FUNCTION_BLOCK JsonDeserializer_TestSuite EXTENDS TcUnit.FB_TestSuite

TestClone();
TestReset();
TestGetArray();
TestGetKeyArray();
TestGetKeyObject();
TestGetObject();
TestTryGetBase64();
TestTryGetBoolWithFalseValue();
TestTryGetBoolWithTrueValue();
TestTryGetByte();
TestTryGetHexAsBytes();
TestTryGetDateTime();
TestTryGetDcTime();
TestTryGetDint();
TestTryGetDword();
TestTryGetFileTime();
TestTryGetInt();
TestTryGetKeyBase64();
TestTryGetKeyBoolWithFalseBoolVariable();
TestTryGetKeyBoolWithTrueBoolVariable();
TestTryGetKeyByte();
TestTryGetKeyHexAsBytes();
TestTryGetKeyDateTime();
TestTryGetKeyDcTime();
TestTryGetKeyDint();
TestTryGetKeyDword();
TestTryGetKeyFileTime();
TestTryGetKeyInt();
TestTryGetKeyLint();
TestTryGetKeyLreal();
TestTryGetKeyLtime();
TestTryGetKeyLword();
TestTryDeserializeKeyToObject();
TestTryDeserializeKeyToObjectFailsWithMissingKey();
TestTryDeserializeKeyToObjectFailsWithInvalidKey();
TestTryGetKeyReal();
TestTryGetKeySint();
TestTryGetKeyString();
TestTryGetKeyTime();
TestTryGetKeyTod();
TestTryGetKeyUdint();
TestTryGetKeyUint();
TestTryGetKeyUlint();
TestTryGetKeyUsint();
TestTryGetKeyWord();
TestTryGetLint();
TestTryGetLreal();
TestTryGetLtime();
TestTryGetLword();
TestTryDeserializeToObject();
TestTryGetReal();
TestTryGetSint();
TestTryGetString();
TestTryGetTime();
TestTryGetTod();
TestTryGetUdint();
TestTryGetUint();
TestTryGetUlint();
TestTryGetUsint();
TestTryGetWord();

METHOD PUBLIC TestClone
VAR
	jsonDeserializer : JsonDeserializer;
	clone : I_Deserializer;
    json : STRING := '{"data":100}';
    out : BYTE;
	feedback : ErrorLogger;
	hasDeserializer : BOOL;
    expected : BYTE := 100;
END_VAR
TEST('TestClone');

// add something to the original 
jsonDeserializer.TryLoad(json);

// deep clone
clone := jsonDeserializer.Clone();

// reset the original
jsonDeserializer.Reset();

// retreive the data from the clone
clone.TryGetKeyByte('data', out, feedback);

// clones are __NEW so must be disposed
clone.Dispose();

AssertEquals(
	Expected := expected,
	Actual := out,
	Message := 'Did not create a deep copy clone'
);

TEST_FINISHED();
END_METHOD

METHOD PUBLIC TestGetArray
VAR
    jsonDeserializer : JsonDeserializer;
	arrayDeserializer : I_Deserializer;
	elementDeserializer : I_Deserializer;
    json : STRING := '[100,200,300]';
    out : BYTE;
	feedback : ErrorLogger;
	hasArrayDeserializer : BOOL;
	hasElementDeserializer : BOOL;
    expected : BYTE := 100;
END_VAR
TEST('TestGetArray');

jsonDeserializer.TryLoad(json);
arrayDeserializer := jsonDeserializer.GetArray();

hasArrayDeserializer := arrayDeserializer <> 0;

IF hasArrayDeserializer THEN
	elementDeserializer := arrayDeserializer.GetElementByIndex(0);
END_IF

AssertTrue(
	Condition := hasArrayDeserializer,
	Message := 'Did not return deserializer for array'
);

hasElementDeserializer := elementDeserializer <> 0;

IF hasElementDeserializer THEN
	elementDeserializer.TryGetByte(out, feedback);
END_IF

AssertTrue(
	Condition := hasElementDeserializer,
	Message := 'Did not return deserializer for element'
);

AssertEquals(
    Expected := expected,
    Actual := out,
    Message := 'Did not produce the expected BYTE value from JSON array'
);

TEST_FINISHED();
END_METHOD

METHOD PUBLIC TestGetKeyArray
VAR
    jsonDeserializer : JsonDeserializer;
	arrayDeserializer : I_Deserializer;
	elementDeserializer : I_Deserializer;
    json : STRING := '{"myArray":[100,200,300]}';
    out : BYTE;
	feedback : ErrorLogger;
	hasArrayDeserializer : BOOL;
	hasElementDeserializer : BOOL;
    expected : BYTE := 100;
END_VAR
TEST('TestGetKeyArray');

jsonDeserializer.TryLoad(json);
arrayDeserializer := jsonDeserializer.GetKeyArray('myArray');

hasArrayDeserializer := arrayDeserializer <> 0;

IF hasArrayDeserializer THEN
	elementDeserializer := arrayDeserializer.GetElementByIndex(0);
END_IF

AssertTrue(
	Condition := hasArrayDeserializer,
	Message := 'Did not return deserializer for array'
);

hasElementDeserializer := elementDeserializer <> 0;

IF hasElementDeserializer THEN
	elementDeserializer.TryGetByte(out, feedback);
END_IF

AssertTrue(
	Condition := hasElementDeserializer,
	Message := 'Did not return deserializer for element'
);

AssertEquals(
    Expected := expected,
    Actual := out,
    Message := 'Did not produce the expected BYTE value from JSON array'
);

TEST_FINISHED();
END_METHOD

METHOD PUBLIC TestGetKeyObject
VAR
    jsonDeserializer : JsonDeserializer;
	objectDeserializer : I_Deserializer;
    json : STRING := '{"data":100}';
    out : BYTE;
	feedback : ErrorLogger;
	hasObjectDeserializer : BOOL;
    expected : BYTE := 100;
END_VAR
TEST('TestGetKeyObject');

jsonDeserializer.TryLoad(json);
objectDeserializer := jsonDeserializer.GetKeyObject('data');

hasObjectDeserializer := objectDeserializer <> 0;

IF hasObjectDeserializer THEN
	objectDeserializer.TryGetByte(out, feedback);
END_IF

AssertTrue(
	Condition := hasObjectDeserializer,
	Message := 'Did not return deserializer for object'
);

AssertEquals(
    Expected := expected,
    Actual := out,
    Message := 'Did not produce the expected BYTE value from JSON'
);

TEST_FINISHED();
END_METHOD

METHOD PUBLIC TestGetObject
VAR
    jsonDeserializer : JsonDeserializer;
	objectDeserializer : I_Deserializer;
    json : STRING := '{"data":100}';
    out : BYTE;
	feedback : ErrorLogger;
	hasObjectDeserializer : BOOL;
    expected : BYTE := 100;
END_VAR
TEST('TestGetObject');

jsonDeserializer.TryLoad(json);
objectDeserializer := jsonDeserializer.GetObject();

hasObjectDeserializer := objectDeserializer <> 0;

IF hasObjectDeserializer THEN
	objectDeserializer.TryGetKeyByte('data',out, feedback);
END_IF

AssertTrue(
	Condition := hasObjectDeserializer,
	Message := 'Did not return deserializer for object'
);

AssertEquals(
    Expected := expected,
    Actual := out,
    Message := 'Did not produce the expected BYTE value from JSON'
);

TEST_FINISHED();
END_METHOD

METHOD PUBLIC TestReset
VAR
	jsonDeserializer : JsonDeserializer;
    json : STRING := '100';
    out : BYTE;
	feedback : ErrorLogger;
    expected : BYTE := 0; 
END_VAR
TEST('TestReset');

jsonDeserializer.TryLoad(json);
jsonDeserializer.Reset();
jsonDeserializer.TryGetByte(out, feedback);

AssertEquals(
	Expected := expected,
	Actual := out,
	Message := 'Did not reset'
);

TEST_FINISHED();
END_METHOD

METHOD PUBLIC TestTryDeserializeKeyToObject
VAR
    jsonDeserializer : JsonDeserializer;
    json : STRING := '{"data":{"Name":"alice","Age":40}}';
    out : MockDeserializableUserObject;
	feedback : ErrorLogger;
    expectedName : STRING := 'alice';
	expectedAge : INT := 40;
	actualName : STRING;
	actualAge : INT;
END_VAR
TEST('TestTryDeserializeKeyToObject');
jsonDeserializer.TryLoad(json);
jsonDeserializer.TryDeserializeKeyToObject('data', out, feedback);

actualName := out.Name;
actualAge := out.Age;

AssertEquals(
    Expected := expectedName,
    Actual := actualName,
    Message := 'Did not produce the expected Object values from JSON'
);

AssertEquals(
    Expected := expectedAge,
    Actual := actualAge,
    Message := 'Did not produce the expected Object values from JSON'
);

TEST_FINISHED();
END_METHOD

METHOD PUBLIC TestTryDeserializeKeyToObjectFailsWithInvalidKey
VAR
    jsonDeserializer : JsonDeserializer;
    json : STRING := '{"data":{"Name":"alice","Age":40}}';
    out : MockDeserializableUserObject;
	feedback : ErrorLogger;
	result : BOOL;
END_VAR
TEST('TestTryDeserializeKeyToObjectFailsWithInvalidKey');
jsonDeserializer.TryLoad(json);
result := jsonDeserializer.TryDeserializeKeyToObject('', out, feedback);

AssertFalse(
	Condition := result,
	Message := 'Try returned true, even though key was invalid present');

TEST_FINISHED();
END_METHOD

METHOD PUBLIC TestTryDeserializeKeyToObjectFailsWithMissingKey
VAR
    jsonDeserializer : JsonDeserializer;
    json : STRING := '{"data":{"Name":"alice","Age":40}}';
    out : MockDeserializableUserObject;
	feedback : ErrorLogger;
	result : BOOL;
END_VAR
TEST('TestTryDeserializeKeyToObjectFailsWithMissingKey');
jsonDeserializer.TryLoad(json);
result := jsonDeserializer.TryDeserializeKeyToObject('test', out, feedback);

AssertFalse(
	Condition := result,
	Message := 'Try returned true, even though key was not present');

TEST_FINISHED();
END_METHOD

METHOD PUBLIC TestTryDeserializeToObject
VAR
    jsonDeserializer : JsonDeserializer;
    json : STRING := '{"Name":"alice","Age":40}';
    out : MockDeserializableUserObject;
	feedback : ErrorLogger;
    expectedName : STRING := 'alice';
	expectedAge : INT := 40;
	actualName : STRING;
	actualAge : INT;
END_VAR
TEST('TestTryDeserializeToObject');

jsonDeserializer.TryLoad(json);
jsonDeserializer.TryDeserializeToObject(out, feedback);

actualName := out.Name;
actualAge := out.Age;

AssertEquals(
    Expected := expectedName,
    Actual := actualName,
    Message := 'Did not produce the expected Object values from JSON'
);

AssertEquals(
    Expected := expectedAge,
    Actual := actualAge,
    Message := 'Did not produce the expected Object values from JSON'
);

TEST_FINISHED();
END_METHOD

METHOD PUBLIC TestTryGetBase64
VAR
	jsonDeserializer : JsonDeserializer;
	json : STRING := '"aGVsbG8="';
	out : ARRAY[0..4] OF BYTE;
	feedback : ErrorLogger;
	expected : ARRAY[0..4] OF BYTE := [104, 101, 108, 108, 111]; 
END_VAR
TEST('TestTryGetBase64');

jsonDeserializer.TryLoad(json);
jsonDeserializer.TryGetBase64(ADR(out), SIZEOF(out), feedback);

AssertEquals(
	Expected := expected,
	Actual := out,
	Message := 'Did not produce the expected Base64 encoded "hello" from JSON'
);

TEST_FINISHED();
END_METHOD

METHOD PUBLIC TestTryGetBoolWithFalseValue
VAR
	jsonDeserializer : JsonDeserializer;
	json : STRING := 'false';
	out : BOOL;
	feedback : ErrorLogger;
	expected : BOOL := FALSE;
END_VAR
TEST('TestTryGetBoolWithFalseValue');

jsonDeserializer.TryLoad(json);
jsonDeserializer.TryGetBool(out, feedback);

AssertEquals(
	Expected := expected,
	Actual := out,
	Message := 'Did not produce the expected JSON string for a false value'
);

TEST_FINISHED();
END_METHOD

METHOD PUBLIC TestTryGetBoolWithTrueValue
VAR
    jsonDeserializer : JsonDeserializer;
    json : STRING := 'true';
    out : BOOL;
	feedback : ErrorLogger;
    expected : BOOL := TRUE; 
END_VAR
TEST('TestTryGetBoolWithTrueValue');

jsonDeserializer.TryLoad(json);
jsonDeserializer.TryGetBool(out, feedback);

AssertEquals(
    Expected := expected,
    Actual := out,
    Message := 'Did not produce the expected true value from JSON'
);

TEST_FINISHED();
END_METHOD

METHOD PUBLIC TestTryGetByte
VAR
    jsonDeserializer : JsonDeserializer;
    json : STRING := '100';
    out : BYTE;
	feedback : ErrorLogger;
    expected : BYTE := 100; 
END_VAR
TEST('TestTryGetByte');

jsonDeserializer.TryLoad(json);
jsonDeserializer.TryGetByte(out, feedback);

AssertEquals(
    Expected := expected,
    Actual := out,
    Message := 'Did not produce the expected BYTE value from JSON'
);

TEST_FINISHED();
END_METHOD

METHOD PUBLIC TestTryGetDateTime
VAR
    jsonDeserializer : JsonDeserializer;
    json : STRING := '"2023-12-30T15:20:00"';
    out : DATE_AND_TIME;
	feedback : ErrorLogger;
    expected : DATE_AND_TIME := DT#2023-12-30-15:20:00; 
END_VAR
TEST('TestTryGetDateTime');

jsonDeserializer.TryLoad(json);
jsonDeserializer.TryGetDateTime(out, feedback);

AssertEquals(
    Expected := expected,
    Actual := out,
    Message := 'Did not produce the expected DATE_AND_TIME value from JSON'
);

TEST_FINISHED();
END_METHOD

METHOD PUBLIC TestTryGetDcTime
VAR
    jsonDeserializer : JsonDeserializer;
    json : STRING := '"2000-01-01T00:00:00.012345678"';
    out : DCTIME;
	feedback : ErrorLogger;
    expected : DCTIME := 12345678;
END_VAR
TEST('TestTryGetDcTime');

jsonDeserializer.TryLoad(json);
jsonDeserializer.TryGetDcTime(out, feedback);

AssertEquals(
    Expected := expected,
    Actual := out,
    Message := 'Did not produce the expected DCTIME value from JSON string'
);

TEST_FINISHED();
END_METHOD

METHOD PUBLIC TestTryGetDint
VAR
    jsonDeserializer : JsonDeserializer;
    json : STRING := '12345';
    out : DINT;
	feedback : ErrorLogger;
    expected : DINT := 12345;
END_VAR
TEST('TestTryGetDint');

jsonDeserializer.TryLoad(json);
jsonDeserializer.TryGetDint(out, feedback);

AssertEquals(
    Expected := expected,
    Actual := out,
    Message := 'Did not produce the expected DINT value from JSON'
);

TEST_FINISHED();
END_METHOD

METHOD PUBLIC TestTryGetDword
VAR
    jsonDeserializer : JsonDeserializer;
    json : STRING := '12345';
    out : DWORD;
	feedback : ErrorLogger;
    expected : DWORD := 12345;
END_VAR
TEST('TestTryGetDword');

jsonDeserializer.TryLoad(json);
jsonDeserializer.TryGetDword(out, feedback);

AssertEquals(
    Expected := expected,
    Actual := out,
    Message := 'Did not produce the expected DWORD value from JSON'
);

TEST_FINISHED();
END_METHOD

METHOD PUBLIC TestTryGetFileTime
VAR
    jsonDeserializer : JsonDeserializer;
    json : STRING := '"1601-01-01T00:00:01.2345678"';
    out : FILETIME;
	feedback : ErrorLogger;
    expected : FILETIME := 12345678; 
END_VAR
TEST('TestTryGetFileTime');

jsonDeserializer.TryLoad(json);
jsonDeserializer.TryGetFileTime(out, feedback);

AssertEquals(
    Expected := expected,
    Actual := out,
    Message := 'Did not produce the expected FILETIME value from JSON'
);

TEST_FINISHED();
END_METHOD

METHOD PUBLIC TestTryGetHexAsBytes
VAR
    jsonDeserializer : JsonDeserializer;
    json : STRING := '"baadf00d"';
    out : ARRAY[0..3] OF BYTE;
	feedback : ErrorLogger;
    expected : ARRAY[0..3] OF BYTE := [16#BA, 16#AD, 16#F0, 16#0D];
END_VAR
TEST('TestTryGetHexAsBytes');

jsonDeserializer.TryLoad(json);
jsonDeserializer.TryGetHexAsBytes(ADR(out), SIZEOF(out), feedback);

AssertEquals(
    Expected := expected,
    Actual := out,
    Message := 'Did not produce the expected binary data from JSON hexadecimal string'
);

TEST_FINISHED();
END_METHOD

METHOD PUBLIC TestTryGetInt
VAR
    jsonDeserializer : JsonDeserializer;
    json : STRING := '12345';
    out : INT;
	feedback : ErrorLogger;
    expected : INT := 12345;
END_VAR
TEST('TestTryGetInt');

jsonDeserializer.TryLoad(json);
jsonDeserializer.TryGetInt(out, feedback);

AssertEquals(
    Expected := expected,
    Actual := out,
    Message := 'Did not produce the expected INT value from JSON'
);

TEST_FINISHED();
END_METHOD

METHOD PUBLIC TestTryGetKeyBase64
VAR
    jsonDeserializer : JsonDeserializer;
    json : STRING := '{"data":"aGVsbG8="}';
    out : ARRAY[0..4] OF BYTE;
	feedback : ErrorLogger;
    expected : ARRAY[0..4] OF BYTE := [104, 101, 108, 108, 111];
END_VAR
TEST('TestTryGetKeyBase64');

jsonDeserializer.TryLoad(json);
jsonDeserializer.TryGetKeyBase64('data', ADR(out), SIZEOF(out), feedback);

AssertEquals(
    Expected := expected,
    Actual := out,
    Message := 'Did not produce the expected binary data from JSON Base64 encoded "hello"'
);

TEST_FINISHED();
END_METHOD

METHOD PUBLIC TestTryGetKeyBoolWithFalseBoolVariable
VAR
    jsonDeserializer : JsonDeserializer;
    json : STRING := '{"data":false}';
    out : BOOL;
	feedback : ErrorLogger;
    expected : BOOL := FALSE;
END_VAR
TEST('TestTryGetKeyBoolWithFalseBoolVariable');

jsonDeserializer.TryLoad(json);
jsonDeserializer.TryGetKeyBool('data', out, feedback);

AssertEquals(
    Expected := expected,
    Actual := out,
    Message := 'Did not produce the expected boolean value from JSON for a false value'
);

TEST_FINISHED();
END_METHOD

METHOD PUBLIC TestTryGetKeyBoolWithTrueBoolVariable
VAR
    jsonDeserializer : JsonDeserializer;
    json : STRING := '{"data":true}';
    out : BOOL;
	feedback : ErrorLogger;
    expected : BOOL := TRUE;
END_VAR
TEST('TestTryGetKeyBoolWithTrueBoolVariable');

jsonDeserializer.TryLoad(json);
jsonDeserializer.TryGetKeyBool('data', out, feedback);

AssertEquals(
    Expected := expected,
    Actual := out,
    Message := 'Did not produce the expected boolean value from JSON for a true value'
);

TEST_FINISHED();
END_METHOD

METHOD PUBLIC TestTryGetKeyByte
VAR
    jsonDeserializer : JsonDeserializer;
    json : STRING := '{"data":100}';
    out : BYTE;
	feedback : ErrorLogger;
    expected : BYTE := 100;
END_VAR
TEST('TestTryGetKeyByte');

jsonDeserializer.TryLoad(json);
jsonDeserializer.TryGetKeyByte('data', out, feedback);

AssertEquals(
    Expected := expected,
    Actual := out,
    Message := 'Did not produce the expected BYTE value from JSON'
);

TEST_FINISHED();
END_METHOD

METHOD PUBLIC TestTryGetKeyDateTime
VAR
    jsonDeserializer : JsonDeserializer;
    json : STRING := '{"data":"2023-12-30T15:20:00"}';
    out : DATE_AND_TIME;
	feedback : ErrorLogger;
    expected : DATE_AND_TIME := DT#2023-12-30-15:20:00;
END_VAR
TEST('TestTryGetKeyDateTime');

jsonDeserializer.TryLoad(json);
jsonDeserializer.TryGetKeyDateTime('data', out, feedback);

AssertEquals(
    Expected := expected,
    Actual := out,
    Message := 'Did not produce the expected DATE_AND_TIME value from JSON'
);

TEST_FINISHED();
END_METHOD

METHOD PUBLIC TestTryGetKeyDcTime
VAR
    jsonDeserializer : JsonDeserializer;
    json : STRING := '{"data":"2000-01-01T00:00:00.012345678"}';
    out : DCTIME;
	feedback : ErrorLogger;
    expected : DCTIME := 12345678;
END_VAR
TEST('TestTryGetKeyDcTime');

jsonDeserializer.TryLoad(json);
jsonDeserializer.TryGetKeyDcTime('data', out, feedback);

AssertEquals(
    Expected := expected,
    Actual := out,
    Message := 'Did not produce the expected DCTIME value from JSON string'
);

TEST_FINISHED();
END_METHOD

METHOD PUBLIC TestTryGetKeyDint
VAR
    jsonDeserializer : JsonDeserializer;
    json : STRING := '{"data":12345}';
    out : DINT;
	feedback : ErrorLogger;
    expected : DINT := 12345;
END_VAR
TEST('TestTryGetKeyDint');

jsonDeserializer.TryLoad(json);
jsonDeserializer.TryGetKeyDint('data', out, feedback);

AssertEquals(
    Expected := expected,
    Actual := out,
    Message := 'Did not produce the expected DINT value from JSON'
);

TEST_FINISHED();
END_METHOD

METHOD PUBLIC TestTryGetKeyDword
VAR
    jsonDeserializer : JsonDeserializer;
    json : STRING := '{"data":12345}';
    out : DWORD;
	feedback : ErrorLogger;
    expected : DWORD := 12345;
END_VAR
TEST('TestTryGetKeyDword');

jsonDeserializer.TryLoad(json);
jsonDeserializer.TryGetKeyDword('data', out, feedback);

AssertEquals(
    Expected := expected,
    Actual := out,
    Message := 'Did not produce the expected DWORD value from JSON'
);

TEST_FINISHED();
END_METHOD

METHOD PUBLIC TestTryGetKeyFileTime
VAR
    jsonDeserializer : JsonDeserializer;
    json : STRING := '{"data":"1601-01-01T00:00:01.2345678"}';
    out : FILETIME;
	feedback : ErrorLogger;
    expected : FILETIME := 12345678;
END_VAR
TEST('TestTryGetKeyFileTime');

jsonDeserializer.TryLoad(json);
jsonDeserializer.TryGetKeyFileTime('data', out, feedback);

AssertEquals(
    Expected := expected,
    Actual := out,
    Message := 'Did not produce the expected FILETIME value from JSON string'
);

TEST_FINISHED();
END_METHOD

METHOD PUBLIC TestTryGetKeyHexAsBytes
VAR
    jsonDeserializer : JsonDeserializer;
    json : STRING := '{"data":"baadf00d"}';
    out : ARRAY[0..3] OF BYTE;
	feedback : ErrorLogger;
    expected : ARRAY[0..3] OF BYTE := [16#BA, 16#AD, 16#F0, 16#0D];
END_VAR
TEST('TestTryGetKeyHexAsBytes');

jsonDeserializer.TryLoad(json);
jsonDeserializer.TryGetKeyHexAsBytes('data', ADR(out), SIZEOF(out), feedback);

AssertEquals(
    Expected := expected,
    Actual := out,
    Message := 'Did not produce the expected binary data from JSON hexadecimal string'
);

TEST_FINISHED();
END_METHOD

METHOD PUBLIC TestTryGetKeyInt
VAR
    jsonDeserializer : JsonDeserializer;
    json : STRING := '{"data":12345}';
    out : INT;
	feedback : ErrorLogger;
    expected : INT := 12345;
END_VAR
TEST('TestTryGetKeyInt');

jsonDeserializer.TryLoad(json);
jsonDeserializer.TryGetKeyInt('data', out, feedback);

AssertEquals(
    Expected := expected,
    Actual := out,
    Message := 'Did not produce the expected INT value from JSON'
);

TEST_FINISHED();
END_METHOD

METHOD PUBLIC TestTryGetKeyLint
VAR
    jsonDeserializer : JsonDeserializer;
    json : STRING := '{"data":9223372036854775807}';
    out : LINT;
	feedback : ErrorLogger;
    expected : LINT := 9223372036854775807;
END_VAR
TEST('TestTryGetKeyLint');

jsonDeserializer.TryLoad(json);
jsonDeserializer.TryGetKeyLint('data', out, feedback);

AssertEquals(
    Expected := expected,
    Actual := out,
    Message := 'Did not produce the expected LINT value from JSON'
);

TEST_FINISHED();
END_METHOD

METHOD PUBLIC TestTryGetKeyLreal
VAR
    jsonDeserializer : JsonDeserializer;
    json : STRING := '{"data":123456.789}';
    out : LREAL;
	feedback : ErrorLogger;
    expected : LREAL := 123456.789;
END_VAR
TEST('TestTryGetKeyLreal');

jsonDeserializer.TryLoad(json);
jsonDeserializer.TryGetKeyLreal('data', out, feedback);

AssertEquals(
    Expected := expected,
    Actual := out,
    Message := 'Did not produce the expected LREAL value from JSON'
);

TEST_FINISHED();
END_METHOD

METHOD PUBLIC TestTryGetKeyLtime
VAR
    jsonDeserializer : JsonDeserializer;
    json : STRING := '{"data":"LTIME#100d2h30m40s500ms600us700ns"}';
    out : LTIME;
	feedback : ErrorLogger;
    expected : LTIME := LTIME#100D2H30M40S500MS600US700NS;
END_VAR
TEST('TestTryGetKeyLtime');

jsonDeserializer.TryLoad(json);
jsonDeserializer.TryGetKeyLtime('data', out, feedback);

AssertEquals(
    Expected := expected,
    Actual := out,
    Message := 'Did not produce the expected LTIME value from JSON string'
);

TEST_FINISHED();
END_METHOD

METHOD PUBLIC TestTryGetKeyLword
VAR
    jsonDeserializer : JsonDeserializer;
    json : STRING := '{"data":9223372036854775807}';
    out : LWORD;
	feedback : ErrorLogger;
    expected : LWORD := 9223372036854775807;
END_VAR
TEST('TestTryGetKeyLword');

jsonDeserializer.TryLoad(json);
jsonDeserializer.TryGetKeyLword('data', out, feedback);

AssertEquals(
    Expected := expected,
    Actual := out,
    Message := 'Did not produce the expected LWORD value from JSON'
);

TEST_FINISHED();
END_METHOD

METHOD PUBLIC TestTryGetKeyReal
VAR
    jsonDeserializer : JsonDeserializer;
    json : STRING := '{"data":123.4}';
    out : REAL;
	feedback : ErrorLogger;
    expected : REAL := 123.4;
END_VAR
TEST('TestTryGetKeyReal');

jsonDeserializer.TryLoad(json);
jsonDeserializer.TryGetKeyReal('data', out, feedback);

AssertEquals(
    Expected := expected,
    Actual := out,
    Message := 'Did not produce the expected REAL value from JSON'
);

TEST_FINISHED();
END_METHOD

METHOD PUBLIC TestTryGetKeySint
VAR
    jsonDeserializer : JsonDeserializer;
    json : STRING := '{"data":123}';
    out : SINT;
	feedback : ErrorLogger;
    expected : SINT := 123;
END_VAR
TEST('TestTryGetKeySint');

jsonDeserializer.TryLoad(json);
jsonDeserializer.TryGetKeySint('data', out, feedback);

AssertEquals(
    Expected := expected,
    Actual := out,
    Message := 'Did not produce the expected SINT value from JSON'
);

TEST_FINISHED();
END_METHOD

METHOD PUBLIC TestTryGetKeyString
VAR
    jsonDeserializer : JsonDeserializer;
    json : STRING := '{"data":"foobar"}';
    out : STRING;
	feedback : ErrorLogger;
    expected : STRING := 'foobar';
END_VAR
TEST('TestTryGetKeyString');

jsonDeserializer.TryLoad(json);
jsonDeserializer.TryGetKeyString('data', out, feedback);

AssertEquals(
    Expected := expected,
    Actual := out,
    Message := 'Did not produce the expected STRING value from JSON'
);

TEST_FINISHED();
END_METHOD

METHOD PUBLIC TestTryGetKeyTime
VAR
    jsonDeserializer : JsonDeserializer;
    json : STRING := '{"data":"T#49d17h2m47s295ms"}';
    out : TIME;
	feedback : ErrorLogger;
    expected : TIME := T#49D17H2M47S295MS;
END_VAR
TEST('TestTryGetKeyTime');

jsonDeserializer.TryLoad(json);
jsonDeserializer.TryGetKeyTime('data', out, feedback);

AssertEquals(
    Expected := expected,
    Actual := out,
    Message := 'Did not produce the expected TIME value from JSON'
);

TEST_FINISHED();
END_METHOD

METHOD PUBLIC TestTryGetKeyTod
VAR
    jsonDeserializer : JsonDeserializer;
    json : STRING := '{"data":"TOD#23:01:23.456"}';
    out : TOD;
	feedback : ErrorLogger;
    expected : TOD := TOD#23:01:23.456;
END_VAR
TEST('TestTryGetKeyTod');

jsonDeserializer.TryLoad(json);
jsonDeserializer.TryGetKeyTod('data', out, feedback);

AssertEquals(
    Expected := expected,
    Actual := out,
    Message := 'Did not produce the expected TOD value from JSON'
);

TEST_FINISHED();
END_METHOD

METHOD PUBLIC TestTryGetKeyUdint
VAR
    jsonDeserializer : JsonDeserializer;
    json : STRING := '{"data":123456}';
    out : UDINT;
	feedback : ErrorLogger;
    expected : UDINT := 123456;
END_VAR
TEST('TestTryGetKeyUdint');

jsonDeserializer.TryLoad(json);
jsonDeserializer.TryGetKeyUdint('data', out, feedback);

AssertEquals(
    Expected := expected,
    Actual := out,
    Message := 'Did not produce the expected UDINT value from JSON'
);

TEST_FINISHED();
END_METHOD

METHOD PUBLIC TestTryGetKeyUint
VAR
    jsonDeserializer : JsonDeserializer;
    json : STRING := '{"data":12345}';
    out : UINT;
	feedback : ErrorLogger;
    expected : UINT := 12345;
END_VAR
TEST('TestTryGetKeyUint');

jsonDeserializer.TryLoad(json);
jsonDeserializer.TryGetKeyUint('data', out, feedback);

AssertEquals(
    Expected := expected,
    Actual := out,
    Message := 'Did not produce the expected UINT value from JSON'
);

TEST_FINISHED();
END_METHOD

METHOD PUBLIC TestTryGetKeyUlint
VAR
    jsonDeserializer : JsonDeserializer;
    json : STRING := '{"data":9223372036854775807}';
    out : ULINT;
	feedback : ErrorLogger;
    expected : ULINT := 9223372036854775807;
END_VAR
TEST('TestTryGetKeyUlint');

jsonDeserializer.TryLoad(json);
jsonDeserializer.TryGetKeyUlint('data', out, feedback);

AssertEquals(
    Expected := expected,
    Actual := out,
    Message := 'Did not produce the expected ULINT value from JSON'
);

TEST_FINISHED();
END_METHOD

METHOD PUBLIC TestTryGetKeyUsint
VAR
    jsonDeserializer : JsonDeserializer;
    json : STRING := '{"data":123}';
    out : USINT;
	feedback : ErrorLogger;
    expected : USINT := 123;
END_VAR
TEST('TestTryGetKeyUsint');

jsonDeserializer.TryLoad(json);
jsonDeserializer.TryGetKeyUsint('data', out, feedback);

AssertEquals(
    Expected := expected,
    Actual := out,
    Message := 'Did not produce the expected USINT value from JSON'
);

TEST_FINISHED();
END_METHOD

METHOD PUBLIC TestTryGetKeyWord
VAR
    jsonDeserializer : JsonDeserializer;
    json : STRING := '{"data":12345}';
    out : WORD;
	feedback : ErrorLogger;
    expected : WORD := 12345;
END_VAR
TEST('TestTryGetKeyWord');

jsonDeserializer.TryLoad(json);
jsonDeserializer.TryGetKeyWord('data', out, feedback);

AssertEquals(
    Expected := expected,
    Actual := out,
    Message := 'Did not produce the expected WORD value from JSON'
);

TEST_FINISHED();
END_METHOD

METHOD PUBLIC TestTryGetLint
VAR
    jsonDeserializer : JsonDeserializer;
    json : STRING := '9223372036854775807';
    out : LINT;
	feedback : ErrorLogger;
    expected : LINT := 9223372036854775807;
END_VAR
TEST('TestTryGetLint');

jsonDeserializer.TryLoad(json);
jsonDeserializer.TryGetLint(out, feedback);

AssertEquals(
    Expected := expected,
    Actual := out,
    Message := 'Did not produce the expected LINT value from JSON'
);

TEST_FINISHED();
END_METHOD

METHOD PUBLIC TestTryGetLreal
VAR
    jsonDeserializer : JsonDeserializer;
    json : STRING := '123456.789';
    out : LREAL;
	feedback : ErrorLogger;
    expected : LREAL := 123456.789;
END_VAR
TEST('TestTryGetLreal');

jsonDeserializer.TryLoad(json);
jsonDeserializer.TryGetLreal(out, feedback);

AssertEquals(
    Expected := expected,
    Actual := out,
    Message := 'Did not produce the expected LREAL value from JSON'
);

TEST_FINISHED();
END_METHOD

METHOD PUBLIC TestTryGetLtime
VAR
    jsonDeserializer : JsonDeserializer;
    json : STRING := '"LTIME#100d2h30m40s500ms600us700ns"';
    out : LTIME;
	feedback : ErrorLogger;
    expected : LTIME := LTIME#100D2H30M40S500MS600US700NS;
END_VAR
TEST('TestTryGetLtime');

jsonDeserializer.TryLoad(json);
jsonDeserializer.TryGetLtime(out, feedback);

AssertEquals(
    Expected := expected,
    Actual := out,
    Message := 'Did not produce the expected LTIME value from JSON string'
);

TEST_FINISHED();
END_METHOD

METHOD PUBLIC TestTryGetLword
VAR
    jsonDeserializer : JsonDeserializer;
    json : STRING := '9223372036854775807';
    out : LWORD;
	feedback : ErrorLogger;
    expected : LWORD := 9223372036854775807;
END_VAR
TEST('TestTryGetLword');

jsonDeserializer.TryLoad(json);
jsonDeserializer.TryGetLword(out, feedback);

AssertEquals(
    Expected := expected,
    Actual := out,
    Message := 'Did not produce the expected LWORD value from JSON'
);

TEST_FINISHED();
END_METHOD

METHOD PUBLIC TestTryGetReal
VAR
    jsonDeserializer : JsonDeserializer;
    json : STRING := '123.4';
    out : REAL;
	feedback : ErrorLogger;
    expected : REAL := 123.4;
END_VAR
TEST('TestTryGetReal');

jsonDeserializer.TryLoad(json);
jsonDeserializer.TryGetReal(out, feedback);

AssertEquals(
    Expected := expected,
    Actual := out,
    Message := 'Did not produce the expected REAL value from JSON'
);

TEST_FINISHED();
END_METHOD

METHOD PUBLIC TestTryGetSint
VAR
    jsonDeserializer : JsonDeserializer;
    json : STRING := '123';
    out : SINT;
	feedback : ErrorLogger;
    expected : SINT := 123;
END_VAR
TEST('TestTryGetSint');

jsonDeserializer.TryLoad(json);
jsonDeserializer.TryGetSint(out, feedback);

AssertEquals(
    Expected := expected,
    Actual := out,
    Message := 'Did not produce the expected SINT value from JSON'
);

TEST_FINISHED();
END_METHOD

METHOD PUBLIC TestTryGetString
VAR
    jsonDeserializer : JsonDeserializer;
    json : STRING := '"foobar"';
    out : STRING;
	feedback : ErrorLogger;
    expected : STRING := 'foobar';
END_VAR
TEST('TestTryGetString');

jsonDeserializer.TryLoad(json);
jsonDeserializer.TryGetString(out, feedback);

AssertEquals(
    Expected := expected,
    Actual := out,
    Message := 'Did not produce the expected STRING value from JSON "foobar"'
);

TEST_FINISHED();
END_METHOD

METHOD PUBLIC TestTryGetTime
VAR
    jsonDeserializer : JsonDeserializer;
    json : STRING := '"T#49d17h2m47s295ms"';
    out : TIME;
	feedback : ErrorLogger;
    expected : TIME := T#49D17H2M47S295MS;
END_VAR
TEST('TestTryGetTime');

jsonDeserializer.TryLoad(json);
jsonDeserializer.TryGetTime(out, feedback);

AssertEquals(
    Expected := expected,
    Actual := out,
    Message := 'Did not produce the expected TIME value from JSON'
);

TEST_FINISHED();
END_METHOD

METHOD PUBLIC TestTryGetTod
VAR
    jsonDeserializer : JsonDeserializer;
    json : STRING := '"TOD#23:01:23.456"';
    out : TOD;
	feedback : ErrorLogger;
    expected : TOD := TOD#23:01:23.456;
END_VAR
TEST('TestTryGetTod');

jsonDeserializer.TryLoad(json);
jsonDeserializer.TryGetTod(out, feedback);

AssertEquals(
    Expected := expected,
    Actual := out,
    Message := 'Did not produce the expected TOD value from JSON string'
);

TEST_FINISHED();
END_METHOD

METHOD PUBLIC TestTryGetUdint
VAR
    jsonDeserializer : JsonDeserializer;
    json : STRING := '123456';
    out : UDINT;
	feedback : ErrorLogger;
    expected : UDINT := 123456;
END_VAR
TEST('TestTryGetUdint');

jsonDeserializer.TryLoad(json);
jsonDeserializer.TryGetUdint(out, feedback);

AssertEquals(
    Expected := expected,
    Actual := out,
    Message := 'Did not produce the expected UDINT value from JSON'
);

TEST_FINISHED();
END_METHOD

METHOD PUBLIC TestTryGetUint
VAR
    jsonDeserializer : JsonDeserializer;
    json : STRING := '12345';
    out : UINT;
	feedback : ErrorLogger;
    expected : UINT := 12345;
END_VAR
TEST('TestTryGetUint');

jsonDeserializer.TryLoad(json);
jsonDeserializer.TryGetUint(out, feedback);

AssertEquals(
    Expected := expected,
    Actual := out,
    Message := 'Did not produce the expected UINT value from JSON'
);

TEST_FINISHED();
END_METHOD

METHOD PUBLIC TestTryGetUlint
VAR
    jsonDeserializer : JsonDeserializer;
    json : STRING := '9223372036854775807';
    out : ULINT;
	feedback : ErrorLogger;
    expected : ULINT := 9223372036854775807;
END_VAR
TEST('TestTryGetUlint');

jsonDeserializer.TryLoad(json);
jsonDeserializer.TryGetUlint(out, feedback);

AssertEquals(
    Expected := expected,
    Actual := out,
    Message := 'Did not produce the expected ULINT value from JSON'
);

TEST_FINISHED();
END_METHOD

METHOD PUBLIC TestTryGetUsint
VAR
    jsonDeserializer : JsonDeserializer;
    json : STRING := '123';
    out : USINT;
	feedback : ErrorLogger;
    expected : USINT := 123;
END_VAR
TEST('TestTryGetUsint');

jsonDeserializer.TryLoad(json);
jsonDeserializer.TryGetUsint(out, feedback);

AssertEquals(
    Expected := expected,
    Actual := out,
    Message := 'Did not produce the expected USINT value from JSON'
);

TEST_FINISHED();
END_METHOD

METHOD PUBLIC TestTryGetWord
VAR
    jsonDeserializer : JsonDeserializer;
    json : STRING := '12345';
    out : WORD;
	feedback : ErrorLogger;
    expected : WORD := 12345;
END_VAR
TEST('TestTryGetWord');

jsonDeserializer.TryLoad(json);
jsonDeserializer.TryGetWord(out, feedback);

AssertEquals(
    Expected := expected,
    Actual := out,
    Message := 'Did not produce the expected WORD value from JSON "12345"'
);

TEST_FINISHED();
END_METHOD

END_FUNCTION_BLOCK

(* stored: Version 1.1.0.1, ProductVersion 3.1.4024.12
   POU JsonDeserializer_TestSuite: Id {6a6abfa1-5855-4e7d-8ca0-8a7a0f357752}, SpecialFunc None
   Method TestClone: Id {6dedfcc2-659f-4018-b014-28d08ef099c6}
   Method TestGetArray: Id {5f994165-719e-45bb-beea-843d26c7afdb}
   Method TestGetKeyArray: Id {cfa7a7fb-c5d2-4334-afc4-a9b46f0f82c4}
   Method TestGetKeyObject: Id {92411e10-8b04-4e3b-8770-1b6bdd927cf2}
   Method TestGetObject: Id {59394502-a2de-468a-9231-09415dbae109}
   Method TestReset: Id {076e52f9-b7af-4fe7-96e2-cd97c20f33bb}
   Method TestTryDeserializeKeyToObject: Id {6bdd018c-a0cb-419e-b993-5b9208606545}
   Method TestTryDeserializeKeyToObjectFailsWithInvalidKey: Id {f948bb94-040d-45c3-95a9-54b66d7cf358}
   Method TestTryDeserializeKeyToObjectFailsWithMissingKey: Id {74da0489-ea90-40b3-bd45-06df3da6f152}
   Method TestTryDeserializeToObject: Id {cfdf2641-abc6-4b40-972a-a68725eed961}
   Method TestTryGetBase64: Id {d358480d-4a2e-4bde-a64c-7495b770c5ca}
   Method TestTryGetBoolWithFalseValue: Id {aff2d09b-332e-4f7b-a0e7-e5ad1ccd40fe}
   Method TestTryGetBoolWithTrueValue: Id {2ccfb697-01e5-4619-bd7e-331f27b04e94}
   Method TestTryGetByte: Id {07569c8c-6350-4ca8-8e1e-ba9d223521f7}
   Method TestTryGetDateTime: Id {240961c8-6fca-4787-9e0f-ec5736a28735}
   Method TestTryGetDcTime: Id {cb824e12-8cf5-4ebe-bc2a-b05a70f21fa7}
   Method TestTryGetDint: Id {53b13c02-d820-4b2e-b61f-8d4b7c29a7e7}
   Method TestTryGetDword: Id {af38fa6b-5636-4534-9df1-fef63a73692d}
   Method TestTryGetFileTime: Id {dd9636d8-64a4-4ee7-acfd-cf00463ecb5e}
   Method TestTryGetHexAsBytes: Id {c2a599df-ac3c-4ed1-8454-8622af99690a}
   Method TestTryGetInt: Id {a2872c73-f4ab-4170-a75e-685b14cf0db6}
   Method TestTryGetKeyBase64: Id {97fe35b1-6498-4644-9956-d27fb147bf9f}
   Method TestTryGetKeyBoolWithFalseBoolVariable: Id {aa2c3d6c-8a51-4910-9612-54be56979458}
   Method TestTryGetKeyBoolWithTrueBoolVariable: Id {597da172-0551-462b-8da3-47fffdbe5c92}
   Method TestTryGetKeyByte: Id {862c1d03-58eb-4314-9470-da7b75f0f373}
   Method TestTryGetKeyDateTime: Id {ac8b20d5-52a6-4f6d-bcb4-0b11208c0039}
   Method TestTryGetKeyDcTime: Id {6ad486ea-b7f8-4dfe-90fa-422976902a4c}
   Method TestTryGetKeyDint: Id {0027c39b-dabf-4ae7-b4ce-ff09911cb35c}
   Method TestTryGetKeyDword: Id {07a1c719-2282-44df-8239-985dc01d7f48}
   Method TestTryGetKeyFileTime: Id {2623a869-2383-4b09-9019-8f6393e98a6d}
   Method TestTryGetKeyHexAsBytes: Id {79d8fcd4-f251-418e-839d-edac98bf07d8}
   Method TestTryGetKeyInt: Id {506b1a2e-e919-4d4c-967e-1d032047db1f}
   Method TestTryGetKeyLint: Id {ae0493e5-00bf-4eb2-8945-0a85f9c9ac9a}
   Method TestTryGetKeyLreal: Id {ce912b60-4e26-4a7c-bb74-797da785d5b6}
   Method TestTryGetKeyLtime: Id {b41069e7-5a8e-4106-96e3-03ed531349ee}
   Method TestTryGetKeyLword: Id {509fa066-4fdf-47a2-a224-4a07533d414f}
   Method TestTryGetKeyReal: Id {5e404505-afce-4f49-b4bd-98aeb35a4d1e}
   Method TestTryGetKeySint: Id {8571cd06-5f66-4cfa-9106-aa3821c5a682}
   Method TestTryGetKeyString: Id {006868e2-91b0-47b7-b426-14b744be906e}
   Method TestTryGetKeyTime: Id {b0de9253-b16a-48d5-9670-e725d90667bc}
   Method TestTryGetKeyTod: Id {516eaafd-8dda-4900-a128-f79542c61fa1}
   Method TestTryGetKeyUdint: Id {d7594fcd-2c0d-4d74-ad97-9999b3f708dd}
   Method TestTryGetKeyUint: Id {1a5a0583-fd5a-49b8-9f35-be6328863a91}
   Method TestTryGetKeyUlint: Id {6a110c25-ea59-4e9e-a50a-4ce6da739d5d}
   Method TestTryGetKeyUsint: Id {1af34b9a-7b86-40c6-9131-2d8f64a8211f}
   Method TestTryGetKeyWord: Id {728bf23c-539e-448a-90b2-f45e56b57dca}
   Method TestTryGetLint: Id {8cd877ad-0b37-4a05-a0bb-d342dff4a405}
   Method TestTryGetLreal: Id {0258eee0-3e2f-489f-8694-0ad15db83892}
   Method TestTryGetLtime: Id {7cd89917-9f3d-4e04-b374-f6c6eceecc73}
   Method TestTryGetLword: Id {729ee115-d16e-4555-8241-5c68cb15bfdf}
   Method TestTryGetReal: Id {adb62929-fcc2-4c5e-956e-2b2bd286e5be}
   Method TestTryGetSint: Id {d64d10bd-4732-4861-b373-2655994ffabe}
   Method TestTryGetString: Id {de2d9c30-7eba-42f6-b352-c094fd4b523f}
   Method TestTryGetTime: Id {0c2e7b28-e014-40cc-a460-dd94d3c3ee78}
   Method TestTryGetTod: Id {6faf7262-46e4-45c3-9a8a-6ae09f936a96}
   Method TestTryGetUdint: Id {68740412-f757-4a34-a690-b7041344e259}
   Method TestTryGetUint: Id {1f8037ba-5128-4983-81f3-fc0498eda1e4}
   Method TestTryGetUlint: Id {b1d912c1-ec8e-44fb-9f82-33bdeaa09ee9}
   Method TestTryGetUsint: Id {017d828c-07ad-4598-b44d-a6071f19b90f}
   Method TestTryGetWord: Id {7dbf9f89-d617-4ad6-b39d-0885404fb414} *)
